PROGRAM MAIN
VAR
END_VAR

RunGrindingWheel();

END_PROGRAM

(* stored: Version 1.1.0.1, ProductVersion 3.1.4020.12
   POU MAIN: Id {3218ea10-728d-4cf7-8834-724c9a906f77}, SpecialFunc None *)
